{attribute addProperty BoxType "ELX1054-0000-0016"}
{attribute addProperty Id "ChannelAT %I*ARRAY[0 ..3] OF BOOL3240"}
{attribute addProperty CRC "1540589371"}
{attribute addProperty SizeInBites "32"}
{attribute addProperty SizeInBytes "4"}
TYPE Input_Type_NC_3EE6969D :
STRUCT
	{attribute addProperty Name "Channel"}
	Channel AT %I* : ARRAY[0 ..3] OF BOOL;
END_STRUCT
END_TYPE

(* stored: Version 1.2.0.0, ProductVersion 3.1.4024.9
   DUT Input_Type_NC_3EE6969D: Id {7289094f-4753-4ee7-b587-ba9a35b7018b} *)
